(*
SPDX-FileCopyrightText: Â© 2026 Oleksandr Tiutyk <trofimich@gmail.com>
SPDX-License-Identifier: MIT
License: https://opensource.org/license/mit
*)

(*!
<summary>Configuration and binding contract for a digital input component.</summary>
<description>
Extends IReadOnlyDigitalInput with hardware IO mapping and contact type mutator.
</description>
*)

INTERFACE IDigitalInput EXTENDS IReadOnlyDigitalInput

(*!
<summary>Binds the component to a raw boolean process image variable.</summary>
<param name="rawValue">Reference to physical boolean input variable '%I*'.</param>
*)
METHOD BindToIO
VAR_INPUT
	rawValue : REFERENCE TO BOOL;
END_VAR
END_METHOD

(*!
<summary>Gets or sets electrical contact configuration.</summary>
*)
{attribute 'monitoring' := 'call'}
PROPERTY ContactType : CONTACT_TYPE
GET
END_GET
SET
END_SET
END_PROPERTY

END_INTERFACE

(* stored: Version 1.1.0.1
   Itf IDigitalInput: Id {3b250580-3a55-494b-88a0-6b2b71c6cc79}
   Method BindToIO: Id {1605f517-9c92-4d01-9cb9-f5bfa59a0a38}
   Property ContactType: Id {6ae1258a-1040-45e8-9622-72a56fb0eb7a}
   Get Get: Id {96d39911-8bb3-49a7-a778-9c9dc0e52a37}
   Set Set: Id {c9a31045-becf-4bee-89ba-60b48648b28a} *)
